Yaskawa INFORM job: DEMO_S1_SHORT.JBI

/JOB
//NAME DEMO_S1_SHORT
//POS
///NPOS 10,0,0,0,0,0
///TOOL 0
///POSTYPE PULSE
///PULSE
C00000=-49979,-47002,-46090,9960,-74251,-36561
C00001=-47961,-50222,-66422,10946,-63821,-38211
C00002=-44873,-45720,-69109,11876,-60210,-39638
C00003=-43636,-44991,-70477,12182,-59191,-40211
C00004=-36544,-30834,-61983,20343,-58160,-44197
C00005=-40089,-35305,-57644,19031,-62047,-42118
C00006=-40533,-78652,-80743,48055,-54716,-46989
C00007=-39940,-68985,-81938,51409,-51263,-49599
C00008=-39906,-64666,-82606,53112,-49632,-50818
C00009=-37288,-48320,-73516,55312,-49386,-52817
//INST
///DATE 2026/08/26 00:00
///ATTR SC,RW
///GROUP1 RB1
NOP
MOVJ C000 VJ=25.00
MOVL C001 V=150.0
MOVL C002 V=150.0
MOVL C003 V=150.0
MOVL C004 V=150.0
MOVL C005 V=150.0
MOVL C006 V=150.0
MOVL C007 V=150.0
MOVL C008 V=150.0
MOVL C009 V=150.0
END
